FUNCTION_BLOCK FB_Backstep
VAR_INPUT
	x1d:REAL;
	x1:REAL;  
	x2:REAL;  
	x3:REAL;  
	Amp:REAL;
	krise:REAL;
	BC_up:REAL;
	BC_down:REAL;
	cyct:REAL;
	k1:REAL;
	f1:REAL;
	f2:REAL;
	k2:REAL;
	k3:REAL;
	L_d:REAL;
	b0:REAL;
	w2:REAL;
	w3:REAL;
	kr1:REAL;
	kr2:REAL;
	beta1:REAL;
	beta2:REAL;
	M:REAL;  
	aw:REAL; 
	daw:REAL; 
	d1:REAL; 
	u_L:REAL; 
END_VAR
VAR_OUTPUT
	z1:REAL;
	a1:REAL;
	ar1:REAL;
	z2:REAL;
	dz2:REAL;
	a2:REAL;
	ar2:REAL;
	z3:REAL;
	u:REAL;
	u_BC:REAL;
	da1:REAL;
	dda1:REAL;
	da2:REAL;
	da2_BC:REAL;
	ed1:REAL;
	ed2:REAL;
END_VAR
VAR
	Feed:REAL:=0;
	L_x1d:REAL:=0;
	LL_x1d:REAL:=0;
	dz1:REAL;
	dx1d:REAL;
	L_dx1d:REAL:=0;
	ddx1d:REAL:=0;
	L_ddx1d:REAL:=0;
	dddx1d:REAL:=0;
	
	sign1:REAL:=0;
	Inte11:REAL:=0;
	Inte12:REAL:=0;
	Inte21:REAL:=0;
	Inte22:REAL:=0;
	
	Tf1:REAL;
	x2f:REAL;
	L_x2f:REAL:=0;
	L_a2:REAL:=0;
	x3f:REAL;
	L_x3f:REAL:=0;
	
	Tf2:REAL;
	
	edx1:REAL;
	ex1:REAL:=0;
	ex2:REAL:=0;
	edx2:REAL;
	edd1:REAL;
	
	ex3:REAL:=0;
	edx3:REAL;
	edd2:REAL;
	
	kr1c:REAL;
	kr2c:REAL;
	beta1c:REAL;
	beta2c:REAL;
END_VAR


edx1:=ex2-3*w2*(ex1-x1);
edx2:=(x3-aw)/M*L_d+ed1-3*w2*w2*(ex1-x1);
edd1:=-w2*w2*w2*(ex1-x1);

edx3:=b0*u_L+ed2-2*w3*(ex3-x3);
edd2:=-w3*w3*(ex3-x3);

ex1:=ex1+edx1*cyct;
ex2:=ex2+edx2*cyct;
ex3:=ex3+edx3*cyct;
ed2:=ed2+edd2*cyct;
ed1:=ed1+edd1*cyct;

z1:=x1-x1d;
dx1d:=(x1d-L_x1d)/cyct;
dz1:=ex2-dx1d;
L_x1d:=x1d;
a1:=dx1d-k1*z1;

z2:=ex2-a1;
ddx1d:=(dx1d-L_dx1d)/cyct;
L_dx1d:=dx1d;
dddx1d:=0*(ddx1d-L_ddx1d)/cyct;
L_ddx1d:=ddx1d;

da1:=ddx1d-k1*(ex2-dx1d);

//变rise1
kr1c:=kr1*EXPT(2.71828,-(Amp-ABS(krise)));
beta1c:=beta1*EXPT(2.71828,-(Amp-ABS(krise)));

ar1:=-M*kr1c*z2-(kr1c*k2*Inte11+beta1c*Inte12);

IF GFY.BC_kr1=0 THEN
	Inte11:=0;
	Inte12:=0;
ELSE
	Inte11:=Inte11+z2*cyct;
	Inte12:=Inte12+Sign(x:=z2)*cyct;
END_IF

a2:=(-k2*z2+M*da1-M*ed1+ar1)/L_d+aw;
//a2:=aw+M*da1-k2*z2+ar1;

dda1:=dddx1d-k1*(edx2-ddx1d);
dz2:=edx2-da1;

z3:=x3-a2;


da2_BC:=(-k2*dz2+M*dda1-M*edd1)/L_d+daw;;


kr2c:=kr2*EXPT(2.71828,-(Amp-ABS(krise)));
beta2c:=beta2*EXPT(2.71828,-(Amp-ABS(krise)));

ar2:=-kr2c*z3-(kr2c*k3*Inte21+beta2c*Inte22);

IF GFY.BC_kr2=0 THEN
	Inte21:=0;
	Inte22:=0;
ELSE
	Inte21:=Inte21+z3*cyct;
	Inte22:=Inte22+Sign(x:=z3)*cyct;
END_IF

u_BC:=(-k3*z3+da2_BC-ed2+ar2)/b0;
u_BC:=saturation(upLMT:=BC_up,downLMT:=BC_down,input:=u_BC);

END_FUNCTION_BLOCK

(* stored: Version 1.1.0.1, ProductVersion 3.1.4024.12
   POU FB_Backstep: Id {4ca8893c-26be-47dd-840b-62eb74c05773}, SpecialFunc None *)
